// TIA Portal project "GP12_V15.1" (V15.1)

(* hardware
DEVICE "S7-1200 station_1"  S7-1200 Station
   slot 0: "Rack_0"  S7-1200 Rack  Rack  V1.0
   slot 1: "A170648_14 CPU  1214C"  CPU 1214C DC/DC/DC  6ES7 214-1AG40-0XB0  V4.2
   slot 2: "DI 8x24VDC_1"  6ES7 221-1BF32-0XB0  V2.0
*)

// ===== PLC "A170648_14 CPU  1214C"  CPU 1214C DC/DC/DC =====

VAR_GLOBAL   // PLC tag table "默认变量表"
   "合格" AT %I0.0 : Bool;
   "不合格" AT %I0.1 : Bool;
   "复位" AT %I0.2 : Bool;
   "急停" AT %I0.3 : Bool;
   "positionCheck" AT %I0.4 : Bool;
   "toolCheck1" AT %I0.5 : Bool;
   "toolCheck2" AT %I0.6 : Bool;
   "toolCheck3" AT %I0.7 : Bool;
   "toolCheck4" AT %I1.0 : Bool;
   "toolCheck5" AT %I1.1 : Bool;
   "toolCheck6" AT %I1.2 : Bool;
   "toolCheck7" AT %I1.3 : Bool;
   "toolCheck8" AT %I1.4 : Bool;
   "toolCheck9" AT %I1.5 : Bool;
   "toolCheck10" AT %I2.0 : Bool;
   "toolCheck11" AT %I2.1 : Bool;
   "toolCheck12" AT %I2.2 : Bool;
   "toolCheck13" AT %I2.3 : Bool;
   "toolCheck14" AT %I2.4 : Bool;
   "toolCheck15" AT %I2.5 : Bool;
   "toolCheck16" AT %I2.6 : Bool;
   "toolCheck17" AT %I2.7 : Bool;
   "启动打标" AT %Q0.0 : Bool;
   "备用(13)" AT %Q0.1 : Bool;
   "三色灯——绿" AT %Q0.2 : Bool;
   "三色灯——黄" AT %Q0.3 : Bool;
   "三色灯——红" AT %Q0.4 : Bool;
   "三色灯——蜂鸣器" AT %Q0.5 : Bool;
   "气源开关" AT %Q0.6 : Bool;
   "备用(14)" AT %Q0.7 : Bool;
   "合格指示灯" AT %Q1.0 : Bool;
   "不合格指示灯" AT %Q1.1 : Bool;
   "防护门上升" AT %Q2.0 : Bool;
   "防护门下降" AT %Q2.1 : Bool;
   "工装移载前进" AT %Q2.2 : Bool;
   "工装移载后退" AT %Q2.3 : Bool;
   "备用(15)" AT %Q2.4 : Bool;
   "备用(16)" AT %Q2.5 : Bool;
   "备用(17)" AT %Q2.6 : Bool;
   "备用(18)" AT %Q2.7 : Bool;
   "检具选取(1)" AT %Q20.0 : Bool;
   "检具选取(2)" AT %Q20.1 : Bool;
   "检具选取(3)" AT %Q20.2 : Bool;
   "检具选取(4)" AT %Q20.3 : Bool;
   "检具选取(5)" AT %Q20.4 : Bool;
   "检具选取(6)" AT %Q20.5 : Bool;
   "检具选取(7)" AT %Q20.6 : Bool;
   "检具拾取(8)" AT %Q20.7 : Bool;
   "检具选取(9)" AT %Q21.0 : Bool;
   "检具选取(10)" AT %Q21.1 : Bool;
   "检具选取(11)" AT %Q21.2 : Bool;
   "检具选取(12)" AT %Q21.3 : Bool;
   "检具选取(13)" AT %Q21.4 : Bool;
   "检具选取(14)" AT %Q21.5 : Bool;
   "检具选取(15)" AT %Q21.6 : Bool;
   "检具选取(16)" AT %Q21.7 : Bool;
   "程序停止" AT %M100.0 : Bool;
   "复位完成" AT %M100.1 : Bool;
   "Clock_1Hz" AT %M0.5 : Bool;
   "AlwaysFALSE" AT %M1.3 : Bool;
   "Clock_Byte" AT %MB0 : Byte;
   "Clock_10Hz" AT %M0.0 : Bool;
   "Clock_5Hz" AT %M0.1 : Bool;
   "Clock_2.5Hz" AT %M0.2 : Bool;
   "Clock_2Hz" AT %M0.3 : Bool;
   "Clock_1.25Hz" AT %M0.4 : Bool;
   "Clock_0.625Hz" AT %M0.6 : Bool;
   "Clock_0.5Hz" AT %M0.7 : Bool;
   "System_Byte" AT %MB1 : Byte;
   "FirstScan" AT %M1.0 : Bool;
   "DiagStatusUpdate" AT %M1.1 : Bool;
   "AlwaysTRUE" AT %M1.2 : Bool;
   "拾取步_9" AT %M202.0 : Bool;
   "拾取步_10" AT %M202.1 : Bool;
   "拾取步_11" AT %M202.2 : Bool;
   "拾取步_12" AT %M202.3 : Bool;
   "拾取步_13" AT %M202.4 : Bool;
   "拾取步_14" AT %M202.5 : Bool;
   "拾取步_15" AT %M202.6 : Bool;
   "拾取步_16" AT %M202.7 : Bool;
   "拾取步_1" AT %M203.0 : Bool;
   "拾取步_2" AT %M203.1 : Bool;
   "拾取步_3" AT %M203.2 : Bool;
   "拾取步_4" AT %M203.3 : Bool;
   "拾取步_5" AT %M203.4 : Bool;
   "拾取步_6" AT %M203.5 : Bool;
   "拾取步_7" AT %M203.6 : Bool;
   "拾取步_8" AT %M203.7 : Bool;
   "拾取步_17" AT %M300.0 : Bool;
   "拾取报错" AT %M400.0 : Bool;
   "检具选取" AT %MW100 : Word;
   "拾取步" AT %MW202 : Word;
   "Tag_1" AT %M306.0 : Bool;
   "Tag_2" AT %M306.1 : Bool;
   "Tag_3" AT %M306.2 : Bool;
   "Tag_4" AT %M306.3 : Bool;
   "Tag_5" AT %M306.4 : Bool;
   "Tag_6" AT %M306.5 : Bool;
   "Tag_7" AT %M306.6 : Bool;
   "Tag_8" AT %M306.7 : Bool;
   "Tag_9" AT %M307.0 : Bool;
   "Tag_10" AT %M307.1 : Bool;
   "Tag_11" AT %M307.2 : Bool;
   "Tag_12" AT %M307.3 : Bool;
   "Tag_13" AT %M307.4 : Bool;
   "Tag_14" AT %M307.5 : Bool;
   "Tag_15" AT %M307.6 : Bool;
   "Tag_16" AT %M307.7 : Bool;
   "拾取开启" AT %MW306 : Word;
END_VAR

DATA_BLOCK "SERVER"   // DB1
{ S7_Optimized_Access := 'FALSE' }
VERSION : 0.1
   VAR
      设备状态 : Int := 0;
      产品型号 : Int := 0;
      错误代码 : Int := 0;
      生产结果 : Int := 0;
      设备编号 : Int := 0;
      检具拾取 : Int;
   END_VAR
BEGIN
END_DATA_BLOCK

DATA_BLOCK "MB_TCON"   // DB2
{ S7_Optimized_Access := 'FALSE' }
VERSION : 0.1
   VAR
      MB_TCON : TCON_IP_v4;
   END_VAR
BEGIN
   MB_TCON.InterfaceId := 64;
   MB_TCON.ID := 1;
   MB_TCON.LocalPort := 502;
   MB_TCON.RemoteAddress.ADDR[1] := 0;
   MB_TCON.RemoteAddress.ADDR[2] := 0;
   MB_TCON.RemoteAddress.ADDR[3] := 0;
   MB_TCON.RemoteAddress.ADDR[4] := 0;
END_DATA_BLOCK

DATA_BLOCK "RESET_DB"   // DB3
{ S7_Optimized_Access := 'TRUE' }
VERSION : 0.1
// stored: InstanceOfName RESET
"RESET"
BEGIN
END_DATA_BLOCK

DATA_BLOCK "ALARM_DB"   // DB4
{ S7_Optimized_Access := 'TRUE' }
VERSION : 0.1
// stored: InstanceOfName ALARM
"ALARM"
BEGIN
END_DATA_BLOCK

DATA_BLOCK "AUTO_DB"   // DB10
{ S7_Optimized_Access := 'TRUE' }
VERSION : 0.1
// stored: InstanceOfName AUTO
"AUTO"
BEGIN
END_DATA_BLOCK

// folder: System blocks/Program resources

DATA_BLOCK "IEC_Timer_0_DB"   // DB5
{ S7_Optimized_Access := 'TRUE' }
AUTHOR : Simatic
FAMILY : IEC
NAME : IEC_TMR
VERSION : 1.0
// stored: InstanceOfName IEC_TIMER
"IEC_TIMER"
BEGIN
END_DATA_BLOCK

DATA_BLOCK "IEC_Timer_0_DB_3"   // DB12
{ S7_Optimized_Access := 'TRUE' }
AUTHOR : Simatic
FAMILY : IEC
NAME : IEC_TMR
VERSION : 1.0
// stored: InstanceOfName IEC_TIMER
"IEC_TIMER"
BEGIN
END_DATA_BLOCK

// folder: (top level)

FUNCTION_BLOCK "ALARM"   // FB1, LAD
{ S7_Optimized_Access := 'TRUE' }
VERSION : 0.1
   VAR
      "Error-ID" : Word;
      TEmp : Array[0..3] of Bool;
      IEC_Timer_0_Instance : TON_TIME;
      IEC_Timer_0_Instance_1 : TON_TIME;
      IEC_Timer_0_Instance_2 : TON_TIME;
      IEC_Timer_0_Instance_3 : TON_TIME;
      IEC_Timer_0_Instance_4 : TON_TIME;
      IEC_Timer_0_Instance_5 : TON_TIME;
      IEC_Timer_0_Instance_6 : TON_TIME;
      IEC_Timer_0_Instance_7 : TON_TIME;
      IEC_Timer_0_Instance_8 : TON_TIME;
      IEC_Timer_0_Instance_9 : TON_TIME;
      IEC_Timer_0_Instance_10 : TON_TIME;
      IEC_Timer_0_Instance_11 : TON_TIME;
      IEC_Timer_0_Instance_12 : TON_TIME;
      IEC_Timer_0_Instance_13 : TON_TIME;
      IEC_Timer_0_Instance_14 : TON_TIME;
      "STEP" : Int;
      IEC_Timer_0_Instance_15 : TON_TIME;
      IEC_Timer_0_Instance_16 : TON_TIME;
      IEC_Timer_0_Instance_17 : TON_TIME;
   END_VAR
BEGIN

REGION Network 1
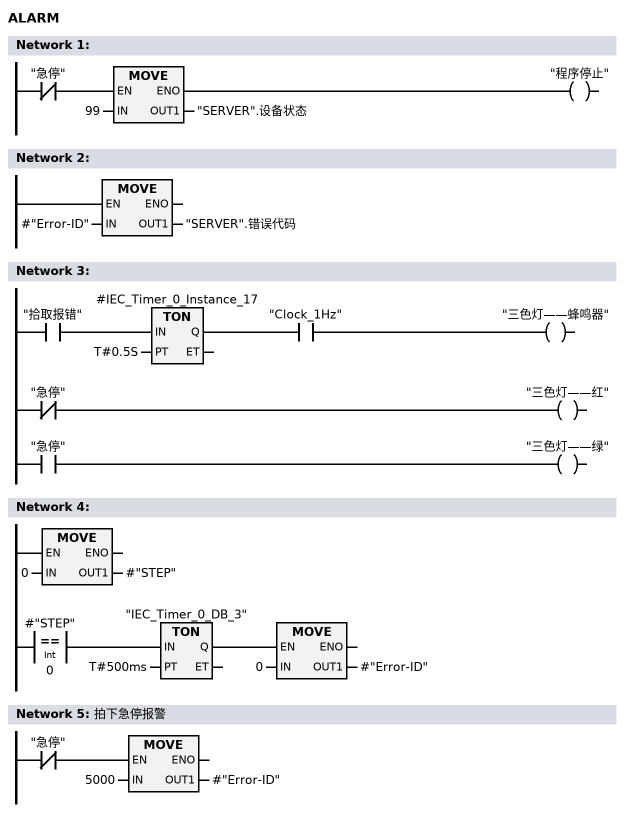
   RUNG wire#powerrail
      I_Contact( "急停" )
      Move(in := 99, out1 => "SERVER".设备状态)
      Coil( "程序停止" )
   END_RUNG
   // the same network as SCL:
   IF NOT "急停" THEN "SERVER".设备状态 := 99; END_IF;
   "程序停止" := NOT "急停";
END_REGION

REGION Network 2
   RUNG wire#powerrail
      Move(in := #"Error-ID", out1 => "SERVER".错误代码)
   END_RUNG
   // the same network as SCL:
   "SERVER".错误代码 := #"Error-ID";
END_REGION

REGION Network 3
   #IEC_Timer_0_Instance_17(IN := "拾取报错", PT := T#0.5S);   // TON
   "三色灯——蜂鸣器" := #IEC_Timer_0_Instance_17.Q AND "Clock_1Hz";
   "三色灯——红" := NOT "急停";
   "三色灯——绿" := "急停";
END_REGION

REGION Network 4
   #"STEP" := 0;
   "IEC_Timer_0_DB_3".TON(IN := #"STEP" = 0, PT := T#500ms);
   IF "IEC_Timer_0_DB_3".Q THEN #"Error-ID" := 0; END_IF;
END_REGION

REGION Network 5: 拍下急停报警
   RUNG wire#powerrail
      I_Contact( "急停" )
      Move(in := 5000, out1 => #"Error-ID")
   END_RUNG
   // the same network as SCL:
   IF NOT "急停" THEN #"Error-ID" := 5000; END_IF;
END_REGION

REGION Network 6: 安全门打开报警
END_REGION

REGION Network 7: 工件未在位启动报警
END_REGION

REGION Network 8: 气源未开报警
END_REGION

REGION Network 9: 工装移栽前进未到位报警
END_REGION

REGION Network 10: 工装移栽未后退报警
END_REGION

REGION Network 11: 防护门未上升报警
END_REGION

REGION Network 12: 防护门为下降报警
END_REGION

REGION Network 13: 1#固定气缸未锁紧报警
END_REGION

REGION Network 14: 1#固定气缸未退回报警
END_REGION

REGION Network 15: 1#机械手未上升报警
END_REGION

REGION Network 16: 1#机械手未下降报警
END_REGION

REGION Network 17: 1#气爪未夹紧到位报警
END_REGION

REGION Network 18: 1#气爪未松开报警
END_REGION

REGION Network 19: 2#机械手未固定锁紧报警
END_REGION

REGION Network 20: 2#固定气缸未退回报警
END_REGION

REGION Network 21: 2#机械手未上升报警
END_REGION

REGION Network 22: 2#机械手未下降报警
END_REGION

REGION Network 23: 2#气爪未夹紧报警
END_REGION

REGION Network 24: 2#气爪未松开报警
END_REGION

REGION Network 25: 激光打码报警
END_REGION
END_FUNCTION_BLOCK

FUNCTION_BLOCK "RESET"   // FB2, LAD
{ S7_Optimized_Access := 'TRUE' }
VERSION : 0.1
   VAR_INPUT
      Stop : Bool;
      Start : Bool;
   END_VAR
   VAR_OUTPUT
      Down : Bool;
   END_VAR
   VAR
      "Step" : Int;
   END_VAR
BEGIN

REGION Network 1
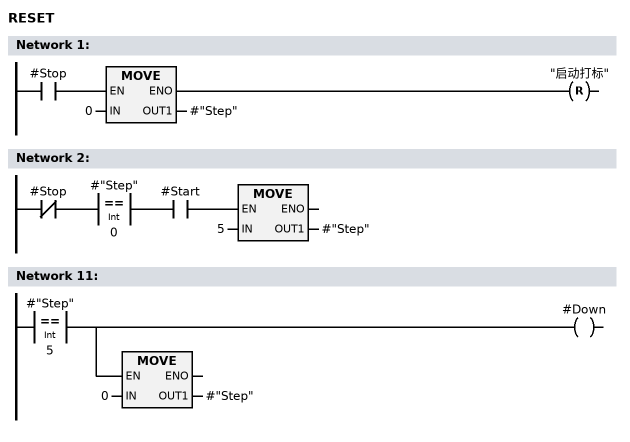
   RUNG wire#powerrail
      Contact( #Stop )
      Move(in := 0, out1 => #"Step")
      R_Coil( "启动打标" )
   END_RUNG
   // the same network as SCL:
   IF #Stop THEN
       #"Step" := 0;
       "启动打标" := FALSE;
   END_IF;
END_REGION

REGION Network 2
   RUNG wire#powerrail
      I_Contact( #Stop )
      { S7_Templates := "SrcType := Int" } EQ_Contact(in1 := #"Step", in2 := 0)
      Contact( #Start )
      Move(in := 5, out1 => #"Step")
   END_RUNG
   // the same network as SCL:
   IF NOT #Stop AND (#"Step" = 0) AND #Start THEN #"Step" := 5; END_IF;
END_REGION

REGION Network 7: 1#气爪松开
END_REGION

REGION Network 8: 2#气爪松开
END_REGION

REGION Network 11
   RUNG wire#powerrail
      { S7_Templates := "SrcType := Int" } EQ_Contact(in1 := #"Step", in2 := 5)
      wire#w1
      Coil( #Down )
   END_RUNG
   RUNG wire#w1
      Move(in := 0, out1 => #"Step")
   END_RUNG
   // the same network as SCL:
   #Down := #"Step" = 5;
   IF #Down THEN #"Step" := 0; END_IF;
END_REGION
END_FUNCTION_BLOCK

FUNCTION_BLOCK "AUTO"   // FB3, LAD
{ S7_Optimized_Access := 'TRUE' }
VERSION : 0.1
   VAR
      IEC_Timer_0_Instance : TON_TIME;
      IEC_Timer_0_Instance_1 : TON_TIME;
   END_VAR
   VAR_TEMP   // added for the SCL form of the ladder/FBD networks
      _w1 : Bool;
   END_VAR
BEGIN

REGION Network 7
   // 复位
END_REGION

REGION Network 8
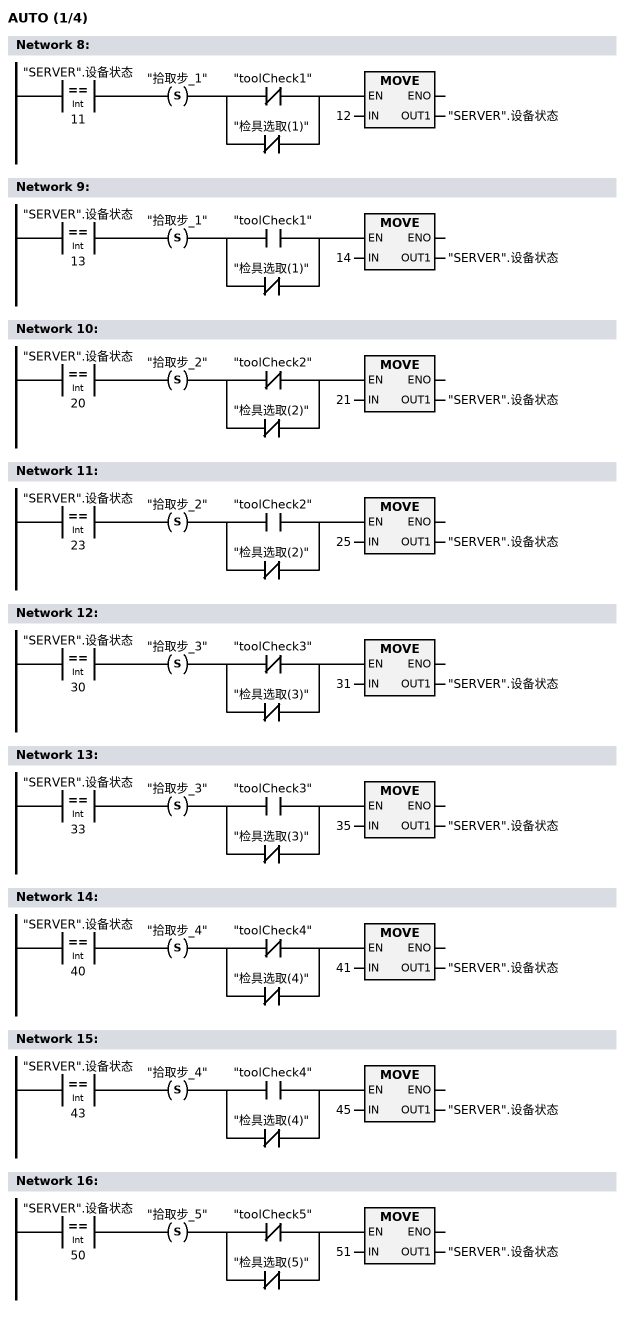
   RUNG wire#powerrail
      { S7_Templates := "SrcType := Int" } EQ_Contact(in1 := "SERVER".设备状态, in2 := 11)
      S_Coil( "拾取步_1" )
      wire#w1
      I_Contact( "toolCheck1" )
      wire#w2
      Move(in := 12, out1 => "SERVER".设备状态)
   END_RUNG
   RUNG wire#w1
      I_Contact( "检具选取(1)" )
   END_RUNG wire#w2
   // the same network as SCL:
   #_w1 := "SERVER".设备状态 = 11;
   IF #_w1 THEN "拾取步_1" := TRUE; END_IF;
   IF #_w1 AND (NOT "toolCheck1" OR NOT "检具选取(1)") THEN "SERVER".设备状态 := 12; END_IF;
END_REGION

REGION Network 9
   RUNG wire#powerrail
      { S7_Templates := "SrcType := Int" } EQ_Contact(in1 := "SERVER".设备状态, in2 := 13)
      S_Coil( "拾取步_1" )
      wire#w1
      Contact( "toolCheck1" )
      wire#w2
      Move(in := 14, out1 => "SERVER".设备状态)
   END_RUNG
   RUNG wire#w1
      I_Contact( "检具选取(1)" )
   END_RUNG wire#w2
   // the same network as SCL:
   #_w1 := "SERVER".设备状态 = 13;
   IF #_w1 THEN "拾取步_1" := TRUE; END_IF;
   IF #_w1 AND ("toolCheck1" OR NOT "检具选取(1)") THEN "SERVER".设备状态 := 14; END_IF;
END_REGION

REGION Network 10
   RUNG wire#powerrail
      { S7_Templates := "SrcType := Int" } EQ_Contact(in1 := "SERVER".设备状态, in2 := 20)
      S_Coil( "拾取步_2" )
      wire#w1
      I_Contact( "toolCheck2" )
      wire#w2
      Move(in := 21, out1 => "SERVER".设备状态)
   END_RUNG
   RUNG wire#w1
      I_Contact( "检具选取(2)" )
   END_RUNG wire#w2
   // the same network as SCL:
   #_w1 := "SERVER".设备状态 = 20;
   IF #_w1 THEN "拾取步_2" := TRUE; END_IF;
   IF #_w1 AND (NOT "toolCheck2" OR NOT "检具选取(2)") THEN "SERVER".设备状态 := 21; END_IF;
END_REGION

REGION Network 11
   RUNG wire#powerrail
      { S7_Templates := "SrcType := Int" } EQ_Contact(in1 := "SERVER".设备状态, in2 := 23)
      S_Coil( "拾取步_2" )
      wire#w1
      Contact( "toolCheck2" )
      wire#w2
      Move(in := 25, out1 => "SERVER".设备状态)
   END_RUNG
   RUNG wire#w1
      I_Contact( "检具选取(2)" )
   END_RUNG wire#w2
   // the same network as SCL:
   #_w1 := "SERVER".设备状态 = 23;
   IF #_w1 THEN "拾取步_2" := TRUE; END_IF;
   IF #_w1 AND ("toolCheck2" OR NOT "检具选取(2)") THEN "SERVER".设备状态 := 25; END_IF;
END_REGION

REGION Network 12
   RUNG wire#powerrail
      { S7_Templates := "SrcType := Int" } EQ_Contact(in1 := "SERVER".设备状态, in2 := 30)
      S_Coil( "拾取步_3" )
      wire#w1
      I_Contact( "toolCheck3" )
      wire#w2
      Move(in := 31, out1 => "SERVER".设备状态)
   END_RUNG
   RUNG wire#w1
      I_Contact( "检具选取(3)" )
   END_RUNG wire#w2
   // the same network as SCL:
   #_w1 := "SERVER".设备状态 = 30;
   IF #_w1 THEN "拾取步_3" := TRUE; END_IF;
   IF #_w1 AND (NOT "toolCheck3" OR NOT "检具选取(3)") THEN "SERVER".设备状态 := 31; END_IF;
END_REGION

REGION Network 13
   RUNG wire#powerrail
      { S7_Templates := "SrcType := Int" } EQ_Contact(in1 := "SERVER".设备状态, in2 := 33)
      S_Coil( "拾取步_3" )
      wire#w1
      Contact( "toolCheck3" )
      wire#w2
      Move(in := 35, out1 => "SERVER".设备状态)
   END_RUNG
   RUNG wire#w1
      I_Contact( "检具选取(3)" )
   END_RUNG wire#w2
   // the same network as SCL:
   #_w1 := "SERVER".设备状态 = 33;
   IF #_w1 THEN "拾取步_3" := TRUE; END_IF;
   IF #_w1 AND ("toolCheck3" OR NOT "检具选取(3)") THEN "SERVER".设备状态 := 35; END_IF;
END_REGION

REGION Network 14
   RUNG wire#powerrail
      { S7_Templates := "SrcType := Int" } EQ_Contact(in1 := "SERVER".设备状态, in2 := 40)
      S_Coil( "拾取步_4" )
      wire#w1
      I_Contact( "toolCheck4" )
      wire#w2
      Move(in := 41, out1 => "SERVER".设备状态)
   END_RUNG
   RUNG wire#w1
      I_Contact( "检具选取(4)" )
   END_RUNG wire#w2
   // the same network as SCL:
   #_w1 := "SERVER".设备状态 = 40;
   IF #_w1 THEN "拾取步_4" := TRUE; END_IF;
   IF #_w1 AND (NOT "toolCheck4" OR NOT "检具选取(4)") THEN "SERVER".设备状态 := 41; END_IF;
END_REGION

REGION Network 15
   RUNG wire#powerrail
      { S7_Templates := "SrcType := Int" } EQ_Contact(in1 := "SERVER".设备状态, in2 := 43)
      S_Coil( "拾取步_4" )
      wire#w1
      Contact( "toolCheck4" )
      wire#w2
      Move(in := 45, out1 => "SERVER".设备状态)
   END_RUNG
   RUNG wire#w1
      I_Contact( "检具选取(4)" )
   END_RUNG wire#w2
   // the same network as SCL:
   #_w1 := "SERVER".设备状态 = 43;
   IF #_w1 THEN "拾取步_4" := TRUE; END_IF;
   IF #_w1 AND ("toolCheck4" OR NOT "检具选取(4)") THEN "SERVER".设备状态 := 45; END_IF;
END_REGION

REGION Network 16
   RUNG wire#powerrail
      { S7_Templates := "SrcType := Int" } EQ_Contact(in1 := "SERVER".设备状态, in2 := 50)
      S_Coil( "拾取步_5" )
      wire#w1
      I_Contact( "toolCheck5" )
      wire#w2
      Move(in := 51, out1 => "SERVER".设备状态)
   END_RUNG
   RUNG wire#w1
      I_Contact( "检具选取(5)" )
   END_RUNG wire#w2
   // the same network as SCL:
   #_w1 := "SERVER".设备状态 = 50;
   IF #_w1 THEN "拾取步_5" := TRUE; END_IF;
   IF #_w1 AND (NOT "toolCheck5" OR NOT "检具选取(5)") THEN "SERVER".设备状态 := 51; END_IF;
END_REGION

REGION Network 17
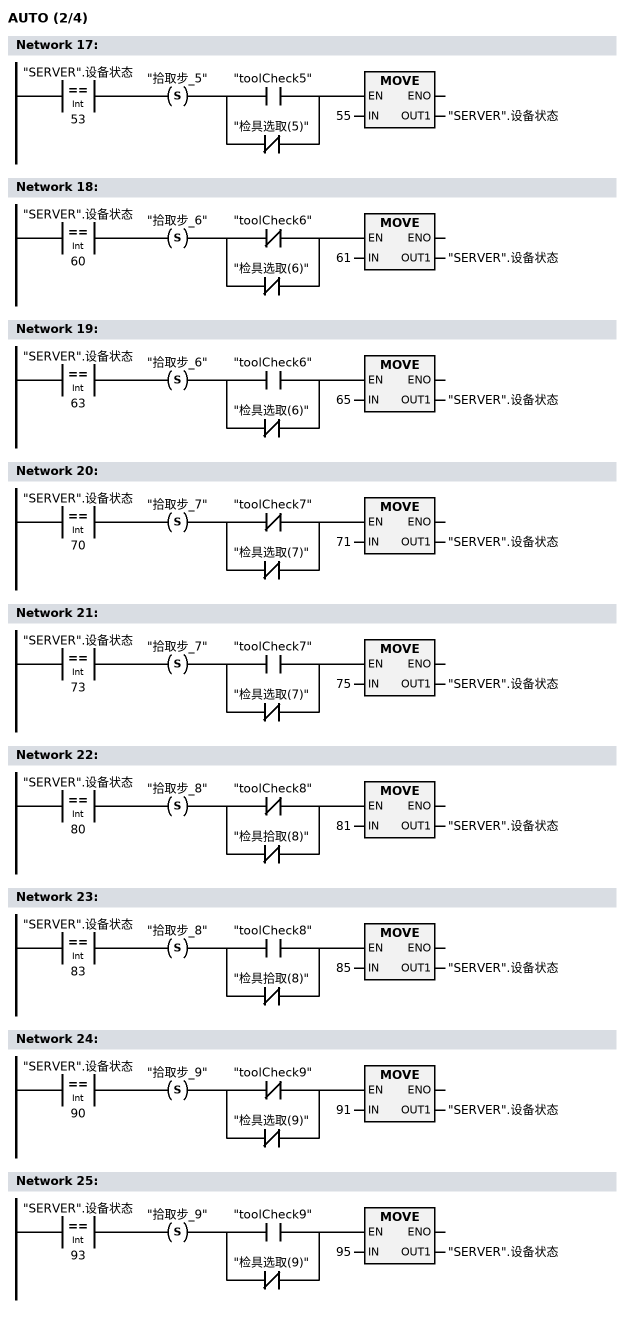
   RUNG wire#powerrail
      { S7_Templates := "SrcType := Int" } EQ_Contact(in1 := "SERVER".设备状态, in2 := 53)
      S_Coil( "拾取步_5" )
      wire#w1
      Contact( "toolCheck5" )
      wire#w2
      Move(in := 55, out1 => "SERVER".设备状态)
   END_RUNG
   RUNG wire#w1
      I_Contact( "检具选取(5)" )
   END_RUNG wire#w2
   // the same network as SCL:
   #_w1 := "SERVER".设备状态 = 53;
   IF #_w1 THEN "拾取步_5" := TRUE; END_IF;
   IF #_w1 AND ("toolCheck5" OR NOT "检具选取(5)") THEN "SERVER".设备状态 := 55; END_IF;
END_REGION

REGION Network 18
   RUNG wire#powerrail
      { S7_Templates := "SrcType := Int" } EQ_Contact(in1 := "SERVER".设备状态, in2 := 60)
      S_Coil( "拾取步_6" )
      wire#w1
      I_Contact( "toolCheck6" )
      wire#w2
      Move(in := 61, out1 => "SERVER".设备状态)
   END_RUNG
   RUNG wire#w1
      I_Contact( "检具选取(6)" )
   END_RUNG wire#w2
   // the same network as SCL:
   #_w1 := "SERVER".设备状态 = 60;
   IF #_w1 THEN "拾取步_6" := TRUE; END_IF;
   IF #_w1 AND (NOT "toolCheck6" OR NOT "检具选取(6)") THEN "SERVER".设备状态 := 61; END_IF;
END_REGION

REGION Network 19
   RUNG wire#powerrail
      { S7_Templates := "SrcType := Int" } EQ_Contact(in1 := "SERVER".设备状态, in2 := 63)
      S_Coil( "拾取步_6" )
      wire#w1
      Contact( "toolCheck6" )
      wire#w2
      Move(in := 65, out1 => "SERVER".设备状态)
   END_RUNG
   RUNG wire#w1
      I_Contact( "检具选取(6)" )
   END_RUNG wire#w2
   // the same network as SCL:
   #_w1 := "SERVER".设备状态 = 63;
   IF #_w1 THEN "拾取步_6" := TRUE; END_IF;
   IF #_w1 AND ("toolCheck6" OR NOT "检具选取(6)") THEN "SERVER".设备状态 := 65; END_IF;
END_REGION

REGION Network 20
   RUNG wire#powerrail
      { S7_Templates := "SrcType := Int" } EQ_Contact(in1 := "SERVER".设备状态, in2 := 70)
      S_Coil( "拾取步_7" )
      wire#w1
      I_Contact( "toolCheck7" )
      wire#w2
      Move(in := 71, out1 => "SERVER".设备状态)
   END_RUNG
   RUNG wire#w1
      I_Contact( "检具选取(7)" )
   END_RUNG wire#w2
   // the same network as SCL:
   #_w1 := "SERVER".设备状态 = 70;
   IF #_w1 THEN "拾取步_7" := TRUE; END_IF;
   IF #_w1 AND (NOT "toolCheck7" OR NOT "检具选取(7)") THEN "SERVER".设备状态 := 71; END_IF;
END_REGION

REGION Network 21
   RUNG wire#powerrail
      { S7_Templates := "SrcType := Int" } EQ_Contact(in1 := "SERVER".设备状态, in2 := 73)
      S_Coil( "拾取步_7" )
      wire#w1
      Contact( "toolCheck7" )
      wire#w2
      Move(in := 75, out1 => "SERVER".设备状态)
   END_RUNG
   RUNG wire#w1
      I_Contact( "检具选取(7)" )
   END_RUNG wire#w2
   // the same network as SCL:
   #_w1 := "SERVER".设备状态 = 73;
   IF #_w1 THEN "拾取步_7" := TRUE; END_IF;
   IF #_w1 AND ("toolCheck7" OR NOT "检具选取(7)") THEN "SERVER".设备状态 := 75; END_IF;
END_REGION

REGION Network 22
   RUNG wire#powerrail
      { S7_Templates := "SrcType := Int" } EQ_Contact(in1 := "SERVER".设备状态, in2 := 80)
      S_Coil( "拾取步_8" )
      wire#w1
      I_Contact( "toolCheck8" )
      wire#w2
      Move(in := 81, out1 => "SERVER".设备状态)
   END_RUNG
   RUNG wire#w1
      I_Contact( "检具拾取(8)" )
   END_RUNG wire#w2
   // the same network as SCL:
   #_w1 := "SERVER".设备状态 = 80;
   IF #_w1 THEN "拾取步_8" := TRUE; END_IF;
   IF #_w1 AND (NOT "toolCheck8" OR NOT "检具拾取(8)") THEN "SERVER".设备状态 := 81; END_IF;
END_REGION

REGION Network 23
   RUNG wire#powerrail
      { S7_Templates := "SrcType := Int" } EQ_Contact(in1 := "SERVER".设备状态, in2 := 83)
      S_Coil( "拾取步_8" )
      wire#w1
      Contact( "toolCheck8" )
      wire#w2
      Move(in := 85, out1 => "SERVER".设备状态)
   END_RUNG
   RUNG wire#w1
      I_Contact( "检具拾取(8)" )
   END_RUNG wire#w2
   // the same network as SCL:
   #_w1 := "SERVER".设备状态 = 83;
   IF #_w1 THEN "拾取步_8" := TRUE; END_IF;
   IF #_w1 AND ("toolCheck8" OR NOT "检具拾取(8)") THEN "SERVER".设备状态 := 85; END_IF;
END_REGION

REGION Network 24
   RUNG wire#powerrail
      { S7_Templates := "SrcType := Int" } EQ_Contact(in1 := "SERVER".设备状态, in2 := 90)
      S_Coil( "拾取步_9" )
      wire#w1
      I_Contact( "toolCheck9" )
      wire#w2
      Move(in := 91, out1 => "SERVER".设备状态)
   END_RUNG
   RUNG wire#w1
      I_Contact( "检具选取(9)" )
   END_RUNG wire#w2
   // the same network as SCL:
   #_w1 := "SERVER".设备状态 = 90;
   IF #_w1 THEN "拾取步_9" := TRUE; END_IF;
   IF #_w1 AND (NOT "toolCheck9" OR NOT "检具选取(9)") THEN "SERVER".设备状态 := 91; END_IF;
END_REGION

REGION Network 25
   RUNG wire#powerrail
      { S7_Templates := "SrcType := Int" } EQ_Contact(in1 := "SERVER".设备状态, in2 := 93)
      S_Coil( "拾取步_9" )
      wire#w1
      Contact( "toolCheck9" )
      wire#w2
      Move(in := 95, out1 => "SERVER".设备状态)
   END_RUNG
   RUNG wire#w1
      I_Contact( "检具选取(9)" )
   END_RUNG wire#w2
   // the same network as SCL:
   #_w1 := "SERVER".设备状态 = 93;
   IF #_w1 THEN "拾取步_9" := TRUE; END_IF;
   IF #_w1 AND ("toolCheck9" OR NOT "检具选取(9)") THEN "SERVER".设备状态 := 95; END_IF;
END_REGION

REGION Network 26
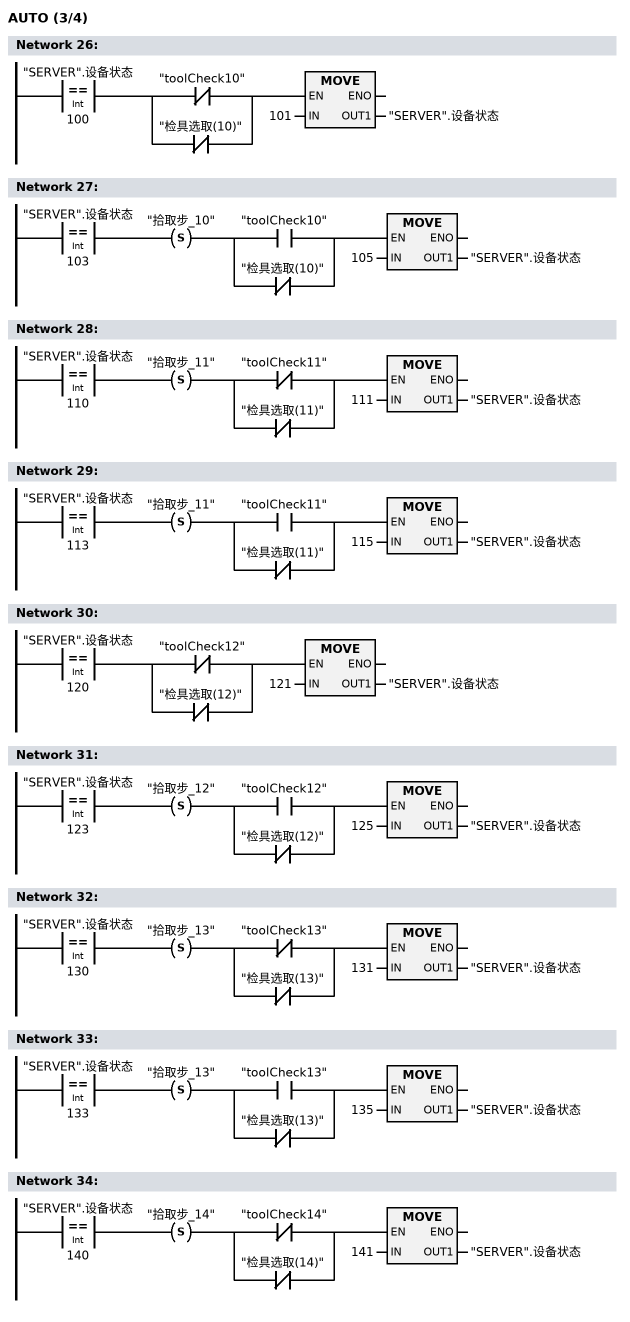
   RUNG wire#powerrail
      { S7_Templates := "SrcType := Int" } EQ_Contact(in1 := "SERVER".设备状态, in2 := 100)
      wire#w1
      I_Contact( "toolCheck10" )
      wire#w2
      Move(in := 101, out1 => "SERVER".设备状态)
   END_RUNG
   RUNG wire#w1
      I_Contact( "检具选取(10)" )
   END_RUNG wire#w2
   // the same network as SCL:
   IF ("SERVER".设备状态 = 100) AND (NOT "toolCheck10" OR NOT "检具选取(10)") THEN "SERVER".设备状态 := 101; END_IF;
END_REGION

REGION Network 27
   RUNG wire#powerrail
      { S7_Templates := "SrcType := Int" } EQ_Contact(in1 := "SERVER".设备状态, in2 := 103)
      S_Coil( "拾取步_10" )
      wire#w1
      Contact( "toolCheck10" )
      wire#w2
      Move(in := 105, out1 => "SERVER".设备状态)
   END_RUNG
   RUNG wire#w1
      I_Contact( "检具选取(10)" )
   END_RUNG wire#w2
   // the same network as SCL:
   #_w1 := "SERVER".设备状态 = 103;
   IF #_w1 THEN "拾取步_10" := TRUE; END_IF;
   IF #_w1 AND ("toolCheck10" OR NOT "检具选取(10)") THEN "SERVER".设备状态 := 105; END_IF;
END_REGION

REGION Network 28
   RUNG wire#powerrail
      { S7_Templates := "SrcType := Int" } EQ_Contact(in1 := "SERVER".设备状态, in2 := 110)
      S_Coil( "拾取步_11" )
      wire#w1
      I_Contact( "toolCheck11" )
      wire#w2
      Move(in := 111, out1 => "SERVER".设备状态)
   END_RUNG
   RUNG wire#w1
      I_Contact( "检具选取(11)" )
   END_RUNG wire#w2
   // the same network as SCL:
   #_w1 := "SERVER".设备状态 = 110;
   IF #_w1 THEN "拾取步_11" := TRUE; END_IF;
   IF #_w1 AND (NOT "toolCheck11" OR NOT "检具选取(11)") THEN "SERVER".设备状态 := 111; END_IF;
END_REGION

REGION Network 29
   RUNG wire#powerrail
      { S7_Templates := "SrcType := Int" } EQ_Contact(in1 := "SERVER".设备状态, in2 := 113)
      S_Coil( "拾取步_11" )
      wire#w1
      Contact( "toolCheck11" )
      wire#w2
      Move(in := 115, out1 => "SERVER".设备状态)
   END_RUNG
   RUNG wire#w1
      I_Contact( "检具选取(11)" )
   END_RUNG wire#w2
   // the same network as SCL:
   #_w1 := "SERVER".设备状态 = 113;
   IF #_w1 THEN "拾取步_11" := TRUE; END_IF;
   IF #_w1 AND ("toolCheck11" OR NOT "检具选取(11)") THEN "SERVER".设备状态 := 115; END_IF;
END_REGION

REGION Network 30
   RUNG wire#powerrail
      { S7_Templates := "SrcType := Int" } EQ_Contact(in1 := "SERVER".设备状态, in2 := 120)
      wire#w1
      I_Contact( "toolCheck12" )
      wire#w2
      Move(in := 121, out1 => "SERVER".设备状态)
   END_RUNG
   RUNG wire#w1
      I_Contact( "检具选取(12)" )
   END_RUNG wire#w2
   // the same network as SCL:
   IF ("SERVER".设备状态 = 120) AND (NOT "toolCheck12" OR NOT "检具选取(12)") THEN "SERVER".设备状态 := 121; END_IF;
END_REGION

REGION Network 31
   RUNG wire#powerrail
      { S7_Templates := "SrcType := Int" } EQ_Contact(in1 := "SERVER".设备状态, in2 := 123)
      S_Coil( "拾取步_12" )
      wire#w1
      Contact( "toolCheck12" )
      wire#w2
      Move(in := 125, out1 => "SERVER".设备状态)
   END_RUNG
   RUNG wire#w1
      I_Contact( "检具选取(12)" )
   END_RUNG wire#w2
   // the same network as SCL:
   #_w1 := "SERVER".设备状态 = 123;
   IF #_w1 THEN "拾取步_12" := TRUE; END_IF;
   IF #_w1 AND ("toolCheck12" OR NOT "检具选取(12)") THEN "SERVER".设备状态 := 125; END_IF;
END_REGION

REGION Network 32
   RUNG wire#powerrail
      { S7_Templates := "SrcType := Int" } EQ_Contact(in1 := "SERVER".设备状态, in2 := 130)
      S_Coil( "拾取步_13" )
      wire#w1
      I_Contact( "toolCheck13" )
      wire#w2
      Move(in := 131, out1 => "SERVER".设备状态)
   END_RUNG
   RUNG wire#w1
      I_Contact( "检具选取(13)" )
   END_RUNG wire#w2
   // the same network as SCL:
   #_w1 := "SERVER".设备状态 = 130;
   IF #_w1 THEN "拾取步_13" := TRUE; END_IF;
   IF #_w1 AND (NOT "toolCheck13" OR NOT "检具选取(13)") THEN "SERVER".设备状态 := 131; END_IF;
END_REGION

REGION Network 33
   RUNG wire#powerrail
      { S7_Templates := "SrcType := Int" } EQ_Contact(in1 := "SERVER".设备状态, in2 := 133)
      S_Coil( "拾取步_13" )
      wire#w1
      Contact( "toolCheck13" )
      wire#w2
      Move(in := 135, out1 => "SERVER".设备状态)
   END_RUNG
   RUNG wire#w1
      I_Contact( "检具选取(13)" )
   END_RUNG wire#w2
   // the same network as SCL:
   #_w1 := "SERVER".设备状态 = 133;
   IF #_w1 THEN "拾取步_13" := TRUE; END_IF;
   IF #_w1 AND ("toolCheck13" OR NOT "检具选取(13)") THEN "SERVER".设备状态 := 135; END_IF;
END_REGION

REGION Network 34
   RUNG wire#powerrail
      { S7_Templates := "SrcType := Int" } EQ_Contact(in1 := "SERVER".设备状态, in2 := 140)
      S_Coil( "拾取步_14" )
      wire#w1
      I_Contact( "toolCheck14" )
      wire#w2
      Move(in := 141, out1 => "SERVER".设备状态)
   END_RUNG
   RUNG wire#w1
      I_Contact( "检具选取(14)" )
   END_RUNG wire#w2
   // the same network as SCL:
   #_w1 := "SERVER".设备状态 = 140;
   IF #_w1 THEN "拾取步_14" := TRUE; END_IF;
   IF #_w1 AND (NOT "toolCheck14" OR NOT "检具选取(14)") THEN "SERVER".设备状态 := 141; END_IF;
END_REGION

REGION Network 35
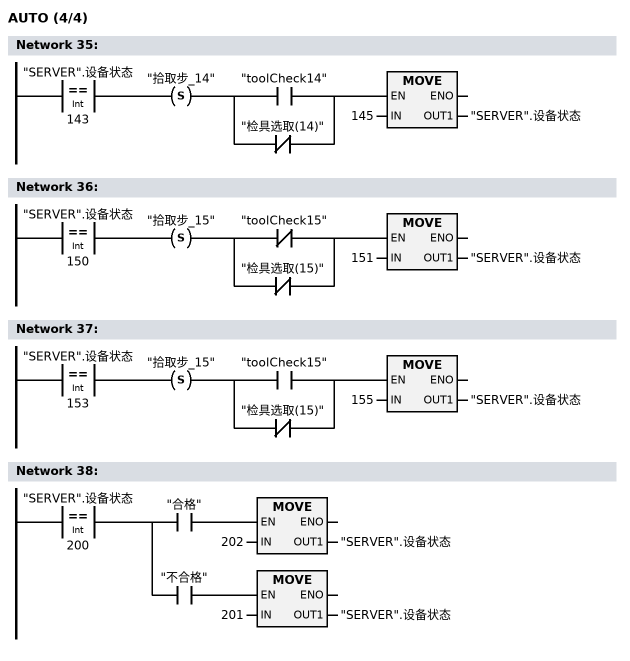
   RUNG wire#powerrail
      { S7_Templates := "SrcType := Int" } EQ_Contact(in1 := "SERVER".设备状态, in2 := 143)
      S_Coil( "拾取步_14" )
      wire#w1
      Contact( "toolCheck14" )
      wire#w2
      Move(in := 145, out1 => "SERVER".设备状态)
   END_RUNG
   RUNG wire#w1
      I_Contact( "检具选取(14)" )
   END_RUNG wire#w2
   // the same network as SCL:
   #_w1 := "SERVER".设备状态 = 143;
   IF #_w1 THEN "拾取步_14" := TRUE; END_IF;
   IF #_w1 AND ("toolCheck14" OR NOT "检具选取(14)") THEN "SERVER".设备状态 := 145; END_IF;
END_REGION

REGION Network 36
   RUNG wire#powerrail
      { S7_Templates := "SrcType := Int" } EQ_Contact(in1 := "SERVER".设备状态, in2 := 150)
      S_Coil( "拾取步_15" )
      wire#w1
      I_Contact( "toolCheck15" )
      wire#w2
      Move(in := 151, out1 => "SERVER".设备状态)
   END_RUNG
   RUNG wire#w1
      I_Contact( "检具选取(15)" )
   END_RUNG wire#w2
   // the same network as SCL:
   #_w1 := "SERVER".设备状态 = 150;
   IF #_w1 THEN "拾取步_15" := TRUE; END_IF;
   IF #_w1 AND (NOT "toolCheck15" OR NOT "检具选取(15)") THEN "SERVER".设备状态 := 151; END_IF;
END_REGION

REGION Network 37
   RUNG wire#powerrail
      { S7_Templates := "SrcType := Int" } EQ_Contact(in1 := "SERVER".设备状态, in2 := 153)
      S_Coil( "拾取步_15" )
      wire#w1
      Contact( "toolCheck15" )
      wire#w2
      Move(in := 155, out1 => "SERVER".设备状态)
   END_RUNG
   RUNG wire#w1
      I_Contact( "检具选取(15)" )
   END_RUNG wire#w2
   // the same network as SCL:
   #_w1 := "SERVER".设备状态 = 153;
   IF #_w1 THEN "拾取步_15" := TRUE; END_IF;
   IF #_w1 AND ("toolCheck15" OR NOT "检具选取(15)") THEN "SERVER".设备状态 := 155; END_IF;
END_REGION

REGION Network 38
   RUNG wire#powerrail
      { S7_Templates := "SrcType := Int" } EQ_Contact(in1 := "SERVER".设备状态, in2 := 200)
      wire#w1
      Contact( "合格" )
      Move(in := 202, out1 => "SERVER".设备状态)
   END_RUNG
   RUNG wire#w1
      Contact( "不合格" )
      Move(in := 201, out1 => "SERVER".设备状态)
   END_RUNG
   // the same network as SCL:
   #_w1 := "SERVER".设备状态 = 200;
   IF #_w1 AND "合格" THEN "SERVER".设备状态 := 202; END_IF;
   IF #_w1 AND "不合格" THEN "SERVER".设备状态 := 201; END_IF;
END_REGION
END_FUNCTION_BLOCK

FUNCTION "拾取" : Void   // FC1, LAD
{ S7_Optimized_Access := 'TRUE' }
VERSION : 0.1
   VAR_INPUT
      拾取0 : Bool;
      拾取1 : Bool;
      拾取2 : Bool;
      拾取3 : Bool;
      拾取4 : Bool;
      拾取5 : Bool;
      拾取6 : Bool;
      拾取7 : Bool;
      拾取8 : Bool;
      拾取9 : Bool;
      拾取10 : Bool;
      拾取11 : Bool;
      拾取12 : Bool;
      拾取13 : Bool;
      拾取14 : Bool;
      拾取15 : Bool;
   END_VAR
   VAR_TEMP
      temp : Word;
   END_VAR
   VAR_TEMP   // added for the SCL form of the ladder/FBD networks
      _w1 : Bool;
   END_VAR
BEGIN

REGION Network 1
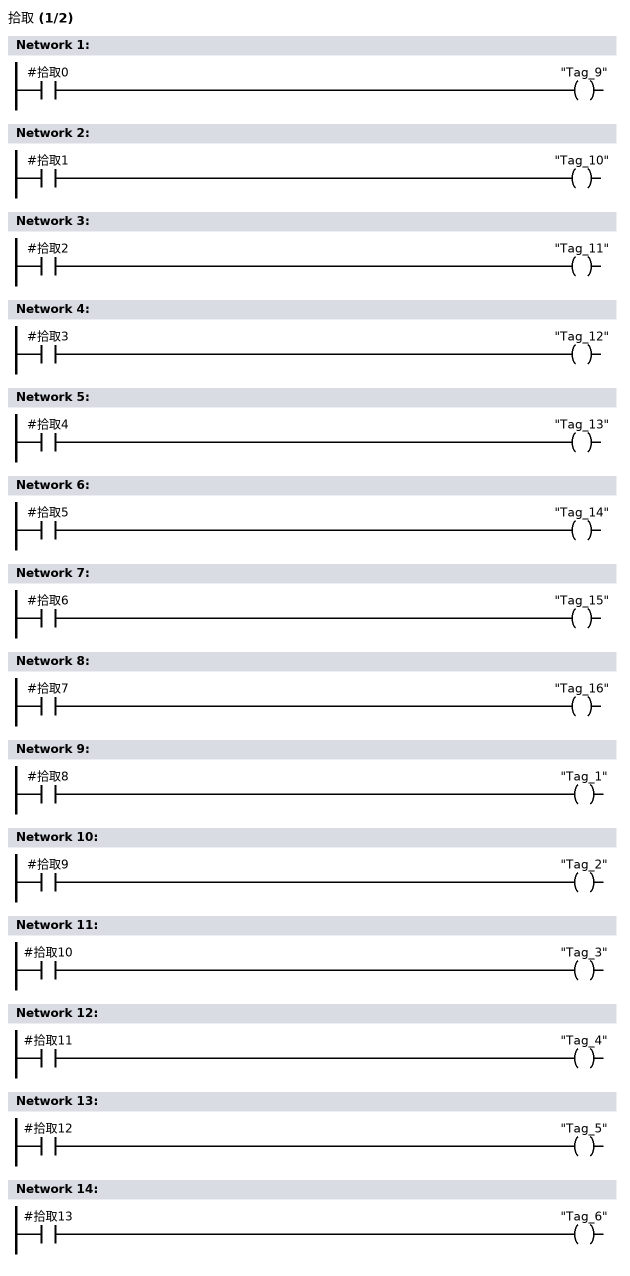
   RUNG wire#powerrail
      Contact( #拾取0 )
      Coil( "Tag_9" )
   END_RUNG
   // the same network as SCL:
   "Tag_9" := #拾取0;
END_REGION

REGION Network 2
   RUNG wire#powerrail
      Contact( #拾取1 )
      Coil( "Tag_10" )
   END_RUNG
   // the same network as SCL:
   "Tag_10" := #拾取1;
END_REGION

REGION Network 3
   RUNG wire#powerrail
      Contact( #拾取2 )
      Coil( "Tag_11" )
   END_RUNG
   // the same network as SCL:
   "Tag_11" := #拾取2;
END_REGION

REGION Network 4
   RUNG wire#powerrail
      Contact( #拾取3 )
      Coil( "Tag_12" )
   END_RUNG
   // the same network as SCL:
   "Tag_12" := #拾取3;
END_REGION

REGION Network 5
   RUNG wire#powerrail
      Contact( #拾取4 )
      Coil( "Tag_13" )
   END_RUNG
   // the same network as SCL:
   "Tag_13" := #拾取4;
END_REGION

REGION Network 6
   RUNG wire#powerrail
      Contact( #拾取5 )
      Coil( "Tag_14" )
   END_RUNG
   // the same network as SCL:
   "Tag_14" := #拾取5;
END_REGION

REGION Network 7
   RUNG wire#powerrail
      Contact( #拾取6 )
      Coil( "Tag_15" )
   END_RUNG
   // the same network as SCL:
   "Tag_15" := #拾取6;
END_REGION

REGION Network 8
   RUNG wire#powerrail
      Contact( #拾取7 )
      Coil( "Tag_16" )
   END_RUNG
   // the same network as SCL:
   "Tag_16" := #拾取7;
END_REGION

REGION Network 9
   RUNG wire#powerrail
      Contact( #拾取8 )
      Coil( "Tag_1" )
   END_RUNG
   // the same network as SCL:
   "Tag_1" := #拾取8;
END_REGION

REGION Network 10
   RUNG wire#powerrail
      Contact( #拾取9 )
      Coil( "Tag_2" )
   END_RUNG
   // the same network as SCL:
   "Tag_2" := #拾取9;
END_REGION

REGION Network 11
   RUNG wire#powerrail
      Contact( #拾取10 )
      Coil( "Tag_3" )
   END_RUNG
   // the same network as SCL:
   "Tag_3" := #拾取10;
END_REGION

REGION Network 12
   RUNG wire#powerrail
      Contact( #拾取11 )
      Coil( "Tag_4" )
   END_RUNG
   // the same network as SCL:
   "Tag_4" := #拾取11;
END_REGION

REGION Network 13
   RUNG wire#powerrail
      Contact( #拾取12 )
      Coil( "Tag_5" )
   END_RUNG
   // the same network as SCL:
   "Tag_5" := #拾取12;
END_REGION

REGION Network 14
   RUNG wire#powerrail
      Contact( #拾取13 )
      Coil( "Tag_6" )
   END_RUNG
   // the same network as SCL:
   "Tag_6" := #拾取13;
END_REGION

REGION Network 15
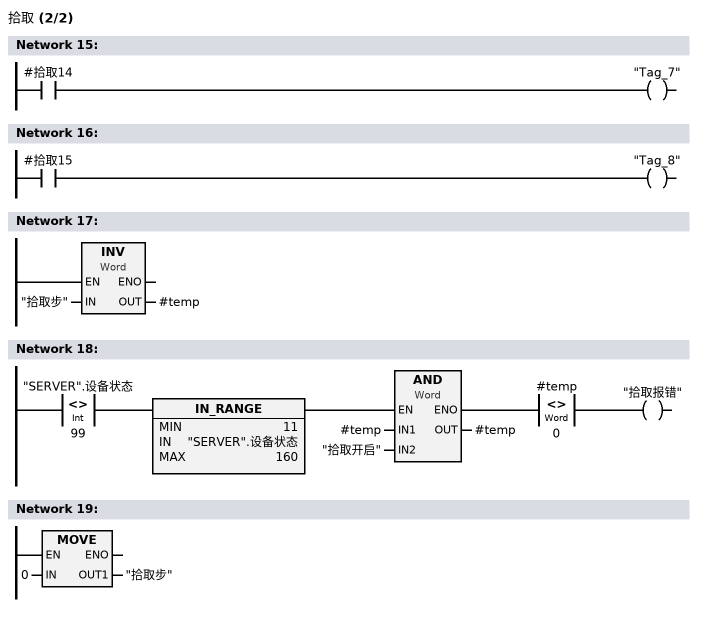
   RUNG wire#powerrail
      Contact( #拾取14 )
      Coil( "Tag_7" )
   END_RUNG
   // the same network as SCL:
   "Tag_7" := #拾取14;
END_REGION

REGION Network 16
   RUNG wire#powerrail
      Contact( #拾取15 )
      Coil( "Tag_8" )
   END_RUNG
   // the same network as SCL:
   "Tag_8" := #拾取15;
END_REGION

REGION Network 17
   RUNG wire#powerrail
      { S7_Templates := "SrcType := Word" } Inv(in := "拾取步", out => #temp)
   END_RUNG
   // the same network as SCL:
   #temp := NOT "拾取步";
END_REGION

REGION Network 18
   RUNG wire#powerrail
      { S7_Templates := "SrcType := Int" } NE_Contact(in1 := "SERVER".设备状态, in2 := 99)
      { S7_Templates := "SrcType := Int" } InRange(min := 11, in := "SERVER".设备状态, max := 160)
      { S7_Templates := "SrcType := Word" } And(in1 := #temp, in2 := "拾取开启", out => #temp)
      { S7_Templates := "SrcType := Word" } NE_Contact(in1 := #temp, in2 := 0)
      Coil( "拾取报错" )
   END_RUNG
   // the same network as SCL:
   #_w1 := ("SERVER".设备状态 <> 99) AND (11 <= "SERVER".设备状态) AND ("SERVER".设备状态 <= 160);
   IF #_w1 THEN #temp := #temp AND "拾取开启"; END_IF;
   "拾取报错" := #_w1 AND (#temp <> 0);
END_REGION

REGION Network 19
   RUNG wire#powerrail
      Move(in := 0, out1 => "拾取步")
   END_RUNG
   // the same network as SCL:
   "拾取步" := 0;
END_REGION
END_FUNCTION

ORGANIZATION_BLOCK "Main"   // OB1, LAD, ProgramCycle
TITLE = "Main Program Sweep (Cycle)"
{ S7_Optimized_Access := 'TRUE' }
VERSION : 0.1
   VAR_INPUT
      Initial_Call : Bool;   // Initial call of this OB
      Remanence : Bool;   // =True, if remanent data are available
   END_VAR
   VAR_TEMP   // added for the SCL form of the ladder/FBD networks
      _w1 : Bool;
   END_VAR
BEGIN

REGION Network 1
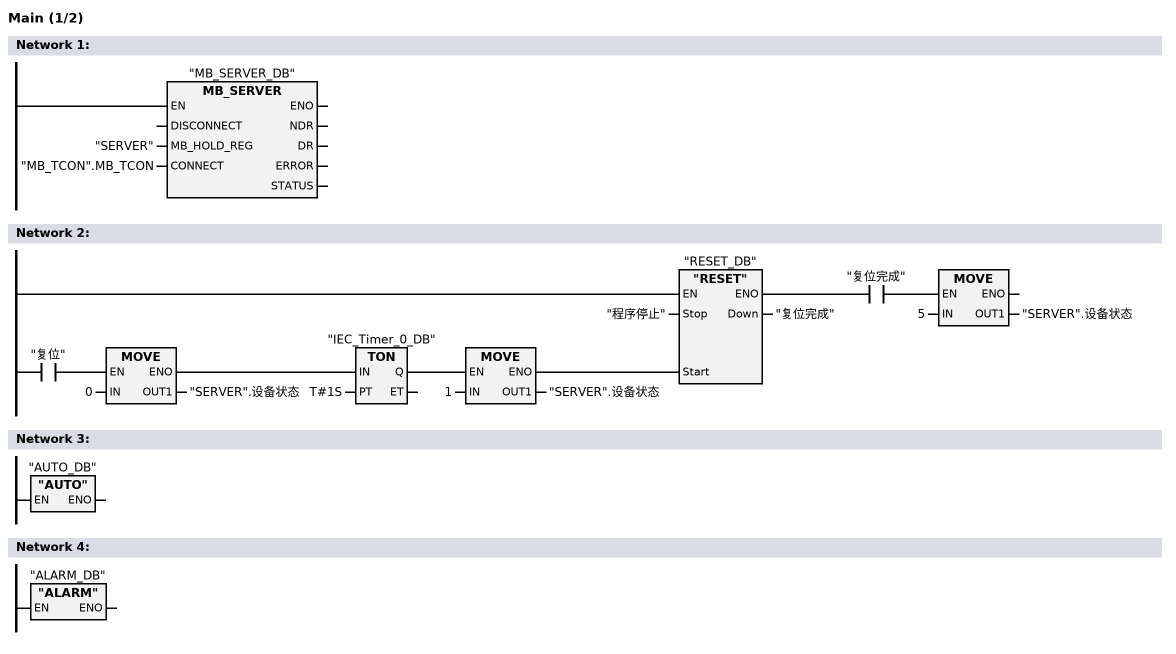
   "MB_SERVER_DB"(MB_HOLD_REG := "SERVER", CONNECT := "MB_TCON".MB_TCON);   // MB_SERVER
END_REGION

REGION Network 2
   IF "复位" THEN "SERVER".设备状态 := 0; END_IF;
   "IEC_Timer_0_DB".TON(IN := "复位", PT := T#1S);
   IF "IEC_Timer_0_DB".Q THEN "SERVER".设备状态 := 1; END_IF;
   "RESET_DB"(Stop := "程序停止", Start := "IEC_Timer_0_DB".Q, Down => "复位完成", ENO => #_w1);   // "RESET"
   IF #_w1 AND "复位完成" THEN "SERVER".设备状态 := 5; END_IF;
END_REGION

REGION Network 3
   RUNG wire#powerrail
      "AUTO_DB"()
   END_RUNG
   // the same network as SCL:
   "AUTO_DB"();   // "AUTO"
END_REGION

REGION Network 4
   RUNG wire#powerrail
      "ALARM_DB"()
   END_RUNG
   // the same network as SCL:
   "ALARM_DB"();   // "ALARM"
END_REGION

REGION Network 5
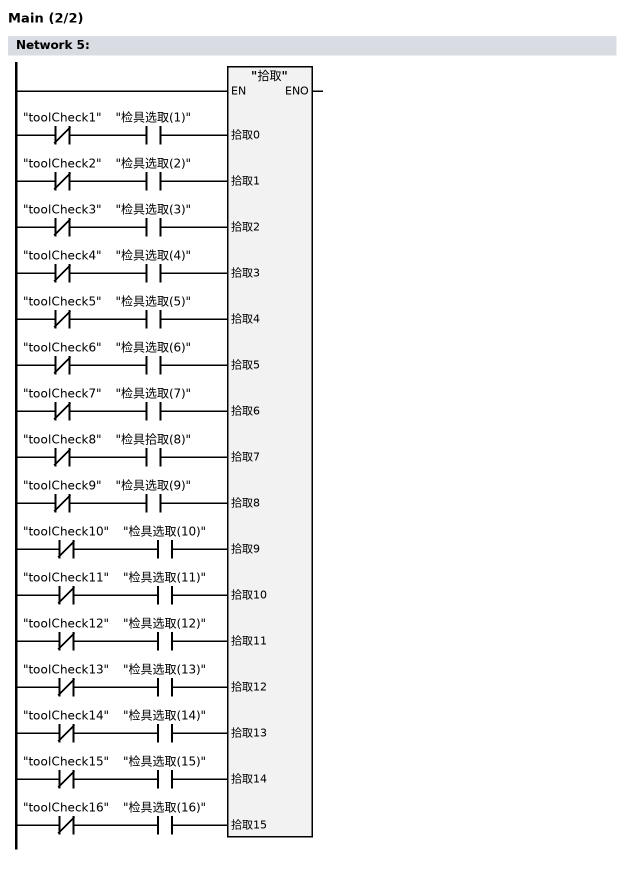
   RUNG wire#powerrail
      "拾取"(拾取0 := wire#w1, 拾取1 := wire#w2, 拾取2 := wire#w3, 拾取3 := wire#w4, 拾取4 := wire#w5, 拾取5 := wire#w6, 拾取6 := wire#w7, 拾取7 := wire#w8, 拾取8 := wire#w9, 拾取9 := wire#w10, 拾取10 := wire#w11, 拾取11 := wire#w12, 拾取12 := wire#w13, 拾取13 := wire#w14, 拾取14 := wire#w15, 拾取15 := wire#w16)
   END_RUNG
   RUNG wire#powerrail
      I_Contact( "toolCheck1" )
      Contact( "检具选取(1)" )
   END_RUNG wire#w1
   RUNG wire#powerrail
      I_Contact( "toolCheck2" )
      Contact( "检具选取(2)" )
   END_RUNG wire#w2
   RUNG wire#powerrail
      I_Contact( "toolCheck3" )
      Contact( "检具选取(3)" )
   END_RUNG wire#w3
   RUNG wire#powerrail
      I_Contact( "toolCheck4" )
      Contact( "检具选取(4)" )
   END_RUNG wire#w4
   RUNG wire#powerrail
      I_Contact( "toolCheck5" )
      Contact( "检具选取(5)" )
   END_RUNG wire#w5
   RUNG wire#powerrail
      I_Contact( "toolCheck6" )
      Contact( "检具选取(6)" )
   END_RUNG wire#w6
   RUNG wire#powerrail
      I_Contact( "toolCheck7" )
      Contact( "检具选取(7)" )
   END_RUNG wire#w7
   RUNG wire#powerrail
      I_Contact( "toolCheck8" )
      Contact( "检具拾取(8)" )
   END_RUNG wire#w8
   RUNG wire#powerrail
      I_Contact( "toolCheck9" )
      Contact( "检具选取(9)" )
   END_RUNG wire#w9
   RUNG wire#powerrail
      I_Contact( "toolCheck10" )
      Contact( "检具选取(10)" )
   END_RUNG wire#w10
   RUNG wire#powerrail
      I_Contact( "toolCheck11" )
      Contact( "检具选取(11)" )
   END_RUNG wire#w11
   RUNG wire#powerrail
      I_Contact( "toolCheck12" )
      Contact( "检具选取(12)" )
   END_RUNG wire#w12
   RUNG wire#powerrail
      I_Contact( "toolCheck13" )
      Contact( "检具选取(13)" )
   END_RUNG wire#w13
   RUNG wire#powerrail
      I_Contact( "toolCheck14" )
      Contact( "检具选取(14)" )
   END_RUNG wire#w14
   RUNG wire#powerrail
      I_Contact( "toolCheck15" )
      Contact( "检具选取(15)" )
   END_RUNG wire#w15
   RUNG wire#powerrail
      I_Contact( "toolCheck16" )
      Contact( "检具选取(16)" )
   END_RUNG wire#w16
   // the same network as SCL:
   "拾取"(拾取0 := NOT "toolCheck1" AND "检具选取(1)",
        拾取1 := NOT "toolCheck2" AND "检具选取(2)",
        拾取2 := NOT "toolCheck3" AND "检具选取(3)",
        拾取3 := NOT "toolCheck4" AND "检具选取(4)",
        拾取4 := NOT "toolCheck5" AND "检具选取(5)",
        拾取5 := NOT "toolCheck6" AND "检具选取(6)",
        拾取6 := NOT "toolCheck7" AND "检具选取(7)",
        拾取7 := NOT "toolCheck8" AND "检具拾取(8)",
        拾取8 := NOT "toolCheck9" AND "检具选取(9)",
        拾取9 := NOT "toolCheck10" AND "检具选取(10)",
        拾取10 := NOT "toolCheck11" AND "检具选取(11)",
        拾取11 := NOT "toolCheck12" AND "检具选取(12)",
        拾取12 := NOT "toolCheck13" AND "检具选取(13)",
        拾取13 := NOT "toolCheck14" AND "检具选取(14)",
        拾取14 := NOT "toolCheck15" AND "检具选取(15)",
        拾取15 := NOT "toolCheck16" AND "检具选取(16)");
END_REGION
END_ORGANIZATION_BLOCK